// TIA Portal V17 export
// export: Created 2023-04-06T15:50:09.30215Z, ExportSetting WithDefaults, DisplayName Totally Integrated Automation Portal, DisplayVersion V17 Update 4, DisplayName TIA Portal Openness, DisplayVersion V17 Update 4, DisplayName TIA Portal Version Control Interface, DisplayVersion V17, DisplayName STEP 7 Professional, DisplayVersion V17 Update 4, DisplayName STEP 7 Safety, DisplayVersion V17, DisplayName WinCC Professional, DisplayVersion V17 Update 4
FUNCTION "LOGIC_PE_1" : Void   // FC7, LAD
{ S7_Optimized_Access := 'TRUE' }
VERSION : 0.1
// stored: AutoNumber true, IsIECCheckEnabled false, SetENOAutomatically false, UDAEnableTagReadback false
   VAR_TEMP
      rVac : Real;
   END_VAR
   VAR_TEMP   // added for the SCL form of the ladder/FBD networks
      _w1 : Bool;
      _w2 : Bool;
      _w3 : Bool;
   END_VAR
BEGIN

REGION Network 1: Write value of Password, P mode and Q mode - to check
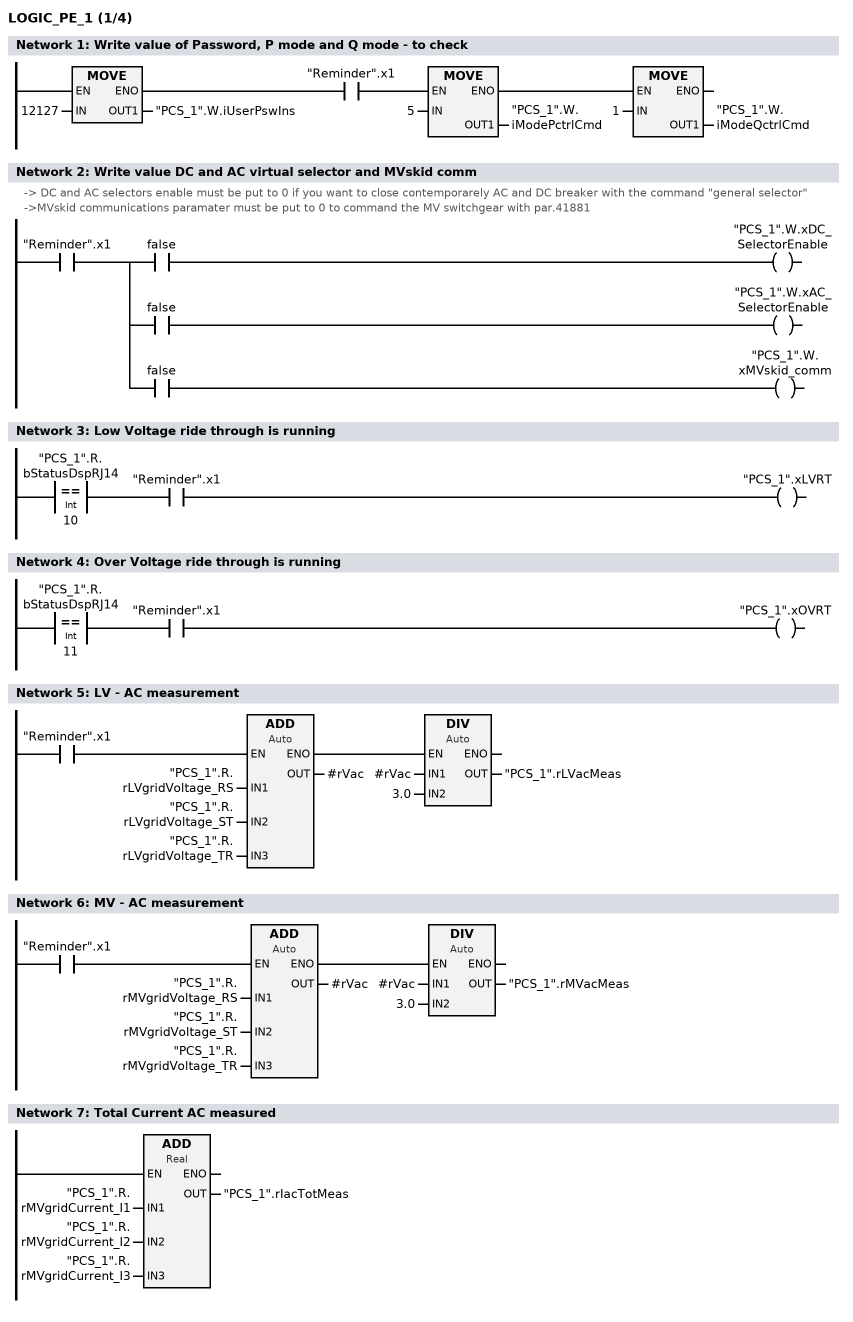
   RUNG wire#powerrail
      Move(in := 12127, out1 => "PCS_1".W.iUserPswIns)
      Contact( "Reminder".x1 )
      Move(in := 5, out1 => "PCS_1".W.iModePctrlCmd)
      Move(in := 1, out1 => "PCS_1".W.iModeQctrlCmd)
   END_RUNG
   // the same network as SCL:
   "PCS_1".W.iUserPswIns := 12127;
   IF "Reminder".x1 THEN
       "PCS_1".W.iModePctrlCmd := 5;
       "PCS_1".W.iModeQctrlCmd := 1;
   END_IF;
END_REGION

REGION Network 2: Write value DC and AC virtual selector and MVskid comm
   // -> DC and AC selectors enable must be put to 0 if you want to close contemporarely AC and DC breaker with the command "general selector"
   // ->MVskid communications paramater must be put to 0 to command the MV switchgear with par.41881
   RUNG wire#powerrail
      Contact( "Reminder".x1 )
      wire#w1
      Contact( false )
      Coil( "PCS_1".W.xDC_SelectorEnable )
   END_RUNG
   RUNG wire#w1
      Contact( false )
      Coil( "PCS_1".W.xAC_SelectorEnable )
   END_RUNG
   RUNG wire#w1
      Contact( false )
      Coil( "PCS_1".W.xMVskid_comm )
   END_RUNG
   // the same network as SCL:
   "PCS_1".W.xDC_SelectorEnable := "Reminder".x1 AND false;
   "PCS_1".W.xAC_SelectorEnable := "Reminder".x1 AND false;
   "PCS_1".W.xMVskid_comm := "Reminder".x1 AND false;
END_REGION

REGION Network 3: Low Voltage ride through is running
   RUNG wire#powerrail
      { S7_Templates := "SrcType := Int" } EQ_Contact(in1 := "PCS_1".R.bStatusDspRJ14, in2 := 10)
      Contact( "Reminder".x1 )
      Coil( "PCS_1".xLVRT )
   END_RUNG
   // the same network as SCL:
   "PCS_1".xLVRT := ("PCS_1".R.bStatusDspRJ14 = 10) AND "Reminder".x1;
END_REGION

REGION Network 4: Over Voltage ride through is running
   RUNG wire#powerrail
      { S7_Templates := "SrcType := Int" } EQ_Contact(in1 := "PCS_1".R.bStatusDspRJ14, in2 := 11)
      Contact( "Reminder".x1 )
      Coil( "PCS_1".xOVRT )
   END_RUNG
   // the same network as SCL:
   "PCS_1".xOVRT := ("PCS_1".R.bStatusDspRJ14 = 11) AND "Reminder".x1;
END_REGION

REGION Network 5: LV - AC measurement
   RUNG wire#powerrail
      Contact( "Reminder".x1 )
      Add(in1 := "PCS_1".R.rLVgridVoltage_RS, in2 := "PCS_1".R.rLVgridVoltage_ST, in3 := "PCS_1".R.rLVgridVoltage_TR, out => #rVac)
      Div(in1 := #rVac, in2 := 3.0, out => "PCS_1".rLVacMeas)
   END_RUNG
   // the same network as SCL:
   IF "Reminder".x1 THEN
       #rVac := "PCS_1".R.rLVgridVoltage_RS + "PCS_1".R.rLVgridVoltage_ST + "PCS_1".R.rLVgridVoltage_TR;
       "PCS_1".rLVacMeas := #rVac / 3.0;
   END_IF;
END_REGION

REGION Network 6: MV - AC measurement
   RUNG wire#powerrail
      Contact( "Reminder".x1 )
      Add(in1 := "PCS_1".R.rMVgridVoltage_RS, in2 := "PCS_1".R.rMVgridVoltage_ST, in3 := "PCS_1".R.rMVgridVoltage_TR, out => #rVac)
      Div(in1 := #rVac, in2 := 3.0, out => "PCS_1".rMVacMeas)
   END_RUNG
   // the same network as SCL:
   IF "Reminder".x1 THEN
       #rVac := "PCS_1".R.rMVgridVoltage_RS + "PCS_1".R.rMVgridVoltage_ST + "PCS_1".R.rMVgridVoltage_TR;
       "PCS_1".rMVacMeas := #rVac / 3.0;
   END_IF;
END_REGION

REGION Network 7: Total Current AC measured
   RUNG wire#powerrail
      { S7_Templates := "SrcType := Real" } Add(in1 := "PCS_1".R.rMVgridCurrent_I1, in2 := "PCS_1".R.rMVgridCurrent_I2, in3 := "PCS_1".R.rMVgridCurrent_I3, out => "PCS_1".rIacTotMeas)
   END_RUNG
   // the same network as SCL:
   "PCS_1".rIacTotMeas := "PCS_1".R.rMVgridCurrent_I1 + "PCS_1".R.rMVgridCurrent_I2 + "PCS_1".R.rMVgridCurrent_I3;
END_REGION

REGION Network 8: Inverter status
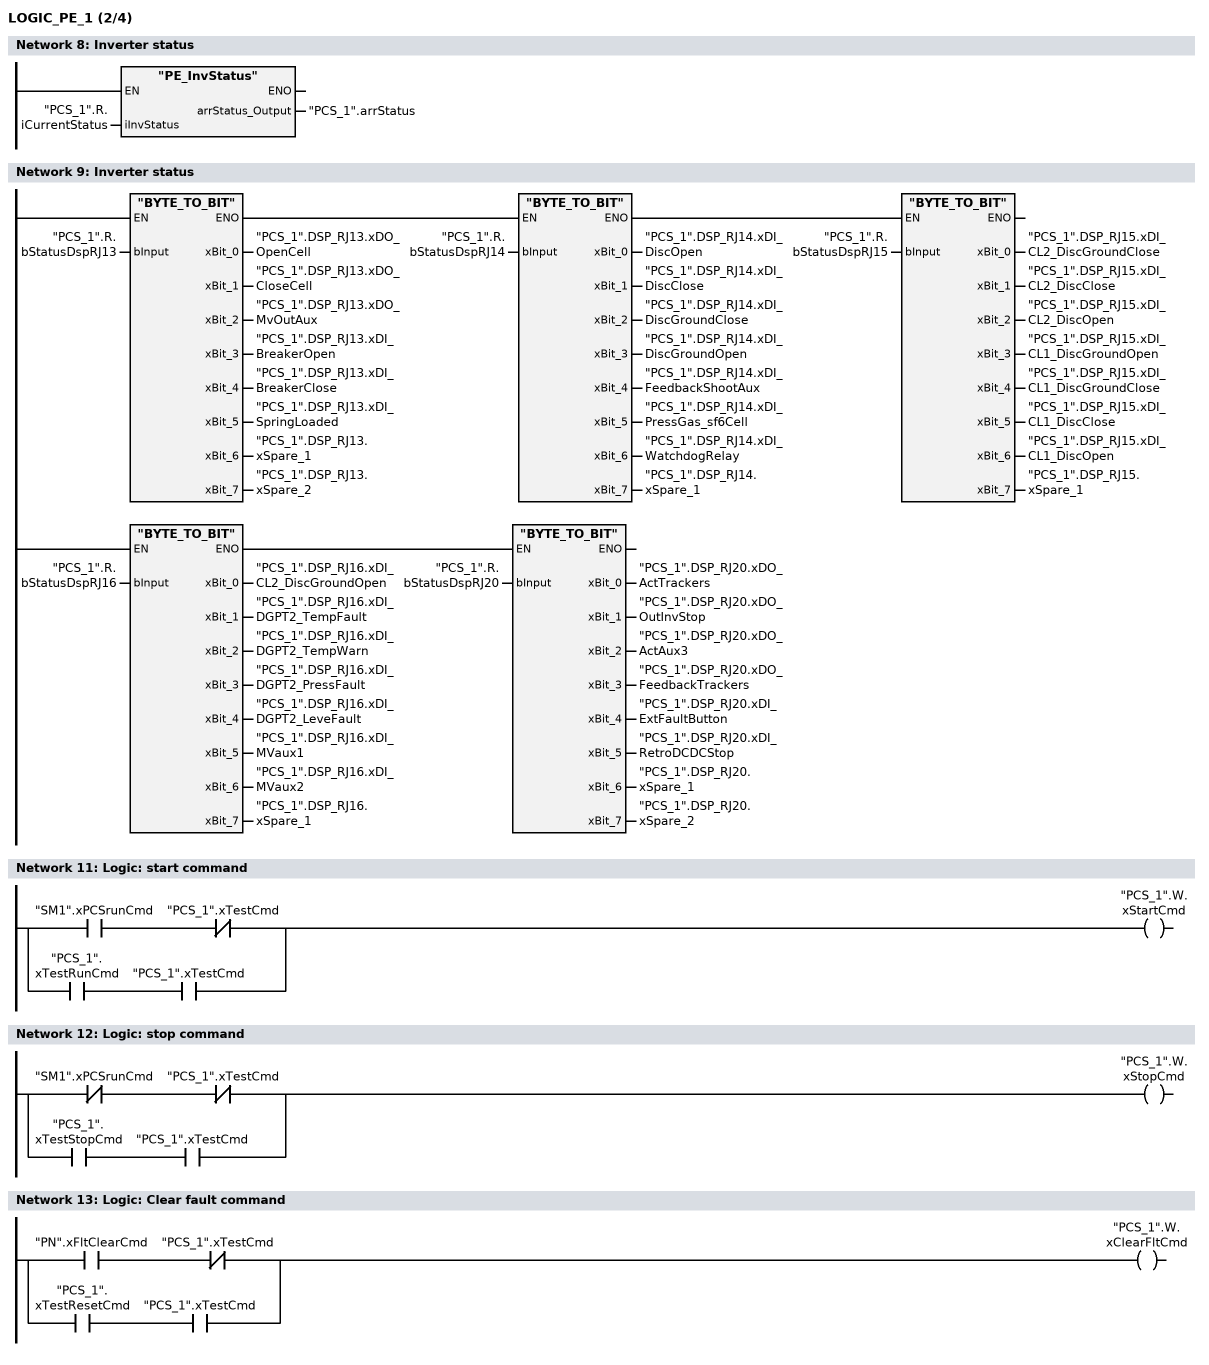
   RUNG wire#powerrail
      "PE_InvStatus"(iInvStatus := "PCS_1".R.iCurrentStatus, arrStatus_Output => "PCS_1".arrStatus)
   END_RUNG
   // the same network as SCL:
   "PE_InvStatus"(iInvStatus := "PCS_1".R.iCurrentStatus, arrStatus_Output => "PCS_1".arrStatus);
END_REGION

REGION Network 9: Inverter status
   RUNG wire#powerrail
      "BYTE_TO_BIT"(bInput := "PCS_1".R.bStatusDspRJ13, xBit_0 => "PCS_1".DSP_RJ13.xDO_OpenCell, xBit_1 => "PCS_1".DSP_RJ13.xDO_CloseCell, xBit_2 => "PCS_1".DSP_RJ13.xDO_MvOutAux, xBit_3 => "PCS_1".DSP_RJ13.xDI_BreakerOpen, xBit_4 => "PCS_1".DSP_RJ13.xDI_BreakerClose, xBit_5 => "PCS_1".DSP_RJ13.xDI_SpringLoaded, xBit_6 => "PCS_1".DSP_RJ13.xSpare_1, xBit_7 => "PCS_1".DSP_RJ13.xSpare_2)
      "BYTE_TO_BIT"(bInput := "PCS_1".R.bStatusDspRJ14, xBit_0 => "PCS_1".DSP_RJ14.xDI_DiscOpen, xBit_1 => "PCS_1".DSP_RJ14.xDI_DiscClose, xBit_2 => "PCS_1".DSP_RJ14.xDI_DiscGroundClose, xBit_3 => "PCS_1".DSP_RJ14.xDI_DiscGroundOpen, xBit_4 => "PCS_1".DSP_RJ14.xDI_FeedbackShootAux, xBit_5 => "PCS_1".DSP_RJ14.xDI_PressGas_sf6Cell, xBit_6 => "PCS_1".DSP_RJ14.xDI_WatchdogRelay, xBit_7 => "PCS_1".DSP_RJ14.xSpare_1)
      "BYTE_TO_BIT"(bInput := "PCS_1".R.bStatusDspRJ15, xBit_0 => "PCS_1".DSP_RJ15.xDI_CL2_DiscGroundClose, xBit_1 => "PCS_1".DSP_RJ15.xDI_CL2_DiscClose, xBit_2 => "PCS_1".DSP_RJ15.xDI_CL2_DiscOpen, xBit_3 => "PCS_1".DSP_RJ15.xDI_CL1_DiscGroundOpen, xBit_4 => "PCS_1".DSP_RJ15.xDI_CL1_DiscGroundClose, xBit_5 => "PCS_1".DSP_RJ15.xDI_CL1_DiscClose, xBit_6 => "PCS_1".DSP_RJ15.xDI_CL1_DiscOpen, xBit_7 => "PCS_1".DSP_RJ15.xSpare_1)
   END_RUNG
   RUNG wire#powerrail
      "BYTE_TO_BIT"(bInput := "PCS_1".R.bStatusDspRJ16, xBit_0 => "PCS_1".DSP_RJ16.xDI_CL2_DiscGroundOpen, xBit_1 => "PCS_1".DSP_RJ16.xDI_DGPT2_TempFault, xBit_2 => "PCS_1".DSP_RJ16.xDI_DGPT2_TempWarn, xBit_3 => "PCS_1".DSP_RJ16.xDI_DGPT2_PressFault, xBit_4 => "PCS_1".DSP_RJ16.xDI_DGPT2_LeveFault, xBit_5 => "PCS_1".DSP_RJ16.xDI_MVaux1, xBit_6 => "PCS_1".DSP_RJ16.xDI_MVaux2, xBit_7 => "PCS_1".DSP_RJ16.xSpare_1)
      "BYTE_TO_BIT"(bInput := "PCS_1".R.bStatusDspRJ20, xBit_0 => "PCS_1".DSP_RJ20.xDO_ActTrackers, xBit_1 => "PCS_1".DSP_RJ20.xDO_OutInvStop, xBit_2 => "PCS_1".DSP_RJ20.xDO_ActAux3, xBit_3 => "PCS_1".DSP_RJ20.xDO_FeedbackTrackers, xBit_4 => "PCS_1".DSP_RJ20.xDI_ExtFaultButton, xBit_5 => "PCS_1".DSP_RJ20.xDI_RetroDCDCStop, xBit_6 => "PCS_1".DSP_RJ20.xSpare_1, xBit_7 => "PCS_1".DSP_RJ20.xSpare_2)
   END_RUNG
   // the same network as SCL:
   "BYTE_TO_BIT"(bInput := "PCS_1".R.bStatusDspRJ13,
                 xBit_0 => "PCS_1".DSP_RJ13.xDO_OpenCell,
                 xBit_1 => "PCS_1".DSP_RJ13.xDO_CloseCell,
                 xBit_2 => "PCS_1".DSP_RJ13.xDO_MvOutAux,
                 xBit_3 => "PCS_1".DSP_RJ13.xDI_BreakerOpen,
                 xBit_4 => "PCS_1".DSP_RJ13.xDI_BreakerClose,
                 xBit_5 => "PCS_1".DSP_RJ13.xDI_SpringLoaded,
                 xBit_6 => "PCS_1".DSP_RJ13.xSpare_1,
                 xBit_7 => "PCS_1".DSP_RJ13.xSpare_2,
                 ENO => #_w1);
   "BYTE_TO_BIT"(EN := #_w1,
                 bInput := "PCS_1".R.bStatusDspRJ14,
                 xBit_0 => "PCS_1".DSP_RJ14.xDI_DiscOpen,
                 xBit_1 => "PCS_1".DSP_RJ14.xDI_DiscClose,
                 xBit_2 => "PCS_1".DSP_RJ14.xDI_DiscGroundClose,
                 xBit_3 => "PCS_1".DSP_RJ14.xDI_DiscGroundOpen,
                 xBit_4 => "PCS_1".DSP_RJ14.xDI_FeedbackShootAux,
                 xBit_5 => "PCS_1".DSP_RJ14.xDI_PressGas_sf6Cell,
                 xBit_6 => "PCS_1".DSP_RJ14.xDI_WatchdogRelay,
                 xBit_7 => "PCS_1".DSP_RJ14.xSpare_1,
                 ENO => #_w2);
   IF #_w2 THEN
       "BYTE_TO_BIT"(bInput := "PCS_1".R.bStatusDspRJ15,
                     xBit_0 => "PCS_1".DSP_RJ15.xDI_CL2_DiscGroundClose,
                     xBit_1 => "PCS_1".DSP_RJ15.xDI_CL2_DiscClose,
                     xBit_2 => "PCS_1".DSP_RJ15.xDI_CL2_DiscOpen,
                     xBit_3 => "PCS_1".DSP_RJ15.xDI_CL1_DiscGroundOpen,
                     xBit_4 => "PCS_1".DSP_RJ15.xDI_CL1_DiscGroundClose,
                     xBit_5 => "PCS_1".DSP_RJ15.xDI_CL1_DiscClose,
                     xBit_6 => "PCS_1".DSP_RJ15.xDI_CL1_DiscOpen,
                     xBit_7 => "PCS_1".DSP_RJ15.xSpare_1);
   END_IF;
   "BYTE_TO_BIT"(bInput := "PCS_1".R.bStatusDspRJ16,
                 xBit_0 => "PCS_1".DSP_RJ16.xDI_CL2_DiscGroundOpen,
                 xBit_1 => "PCS_1".DSP_RJ16.xDI_DGPT2_TempFault,
                 xBit_2 => "PCS_1".DSP_RJ16.xDI_DGPT2_TempWarn,
                 xBit_3 => "PCS_1".DSP_RJ16.xDI_DGPT2_PressFault,
                 xBit_4 => "PCS_1".DSP_RJ16.xDI_DGPT2_LeveFault,
                 xBit_5 => "PCS_1".DSP_RJ16.xDI_MVaux1,
                 xBit_6 => "PCS_1".DSP_RJ16.xDI_MVaux2,
                 xBit_7 => "PCS_1".DSP_RJ16.xSpare_1,
                 ENO => #_w3);
   IF #_w3 THEN
       "BYTE_TO_BIT"(bInput := "PCS_1".R.bStatusDspRJ20,
                     xBit_0 => "PCS_1".DSP_RJ20.xDO_ActTrackers,
                     xBit_1 => "PCS_1".DSP_RJ20.xDO_OutInvStop,
                     xBit_2 => "PCS_1".DSP_RJ20.xDO_ActAux3,
                     xBit_3 => "PCS_1".DSP_RJ20.xDO_FeedbackTrackers,
                     xBit_4 => "PCS_1".DSP_RJ20.xDI_ExtFaultButton,
                     xBit_5 => "PCS_1".DSP_RJ20.xDI_RetroDCDCStop,
                     xBit_6 => "PCS_1".DSP_RJ20.xSpare_1,
                     xBit_7 => "PCS_1".DSP_RJ20.xSpare_2);
   END_IF;
END_REGION

REGION Network 11: Logic: start command
   RUNG wire#powerrail
      Contact( "SM1".xPCSrunCmd )
      I_Contact( "PCS_1".xTestCmd )
      wire#w1
      Coil( "PCS_1".W.xStartCmd )
   END_RUNG
   RUNG wire#powerrail
      Contact( "PCS_1".xTestRunCmd )
      Contact( "PCS_1".xTestCmd )
   END_RUNG wire#w1
   // the same network as SCL:
   "PCS_1".W.xStartCmd := ("SM1".xPCSrunCmd AND NOT "PCS_1".xTestCmd) OR ("PCS_1".xTestRunCmd AND "PCS_1".xTestCmd);
END_REGION

REGION Network 12: Logic: stop command
   RUNG wire#powerrail
      I_Contact( "SM1".xPCSrunCmd )
      I_Contact( "PCS_1".xTestCmd )
      wire#w1
      Coil( "PCS_1".W.xStopCmd )
   END_RUNG
   RUNG wire#powerrail
      Contact( "PCS_1".xTestStopCmd )
      Contact( "PCS_1".xTestCmd )
   END_RUNG wire#w1
   // the same network as SCL:
   "PCS_1".W.xStopCmd := (NOT "SM1".xPCSrunCmd AND NOT "PCS_1".xTestCmd) OR ("PCS_1".xTestStopCmd AND "PCS_1".xTestCmd);
END_REGION

REGION Network 13: Logic: Clear fault command
   RUNG wire#powerrail
      Contact( "PN".xFltClearCmd )
      I_Contact( "PCS_1".xTestCmd )
      wire#w1
      Coil( "PCS_1".W.xClearFltCmd )
   END_RUNG
   RUNG wire#powerrail
      Contact( "PCS_1".xTestResetCmd )
      Contact( "PCS_1".xTestCmd )
   END_RUNG wire#w1
   // the same network as SCL:
   "PCS_1".W.xClearFltCmd := ("PN".xFltClearCmd AND NOT "PCS_1".xTestCmd) OR ("PCS_1".xTestResetCmd AND "PCS_1".xTestCmd);
END_REGION

REGION Network 14: Logic : PPC enable command
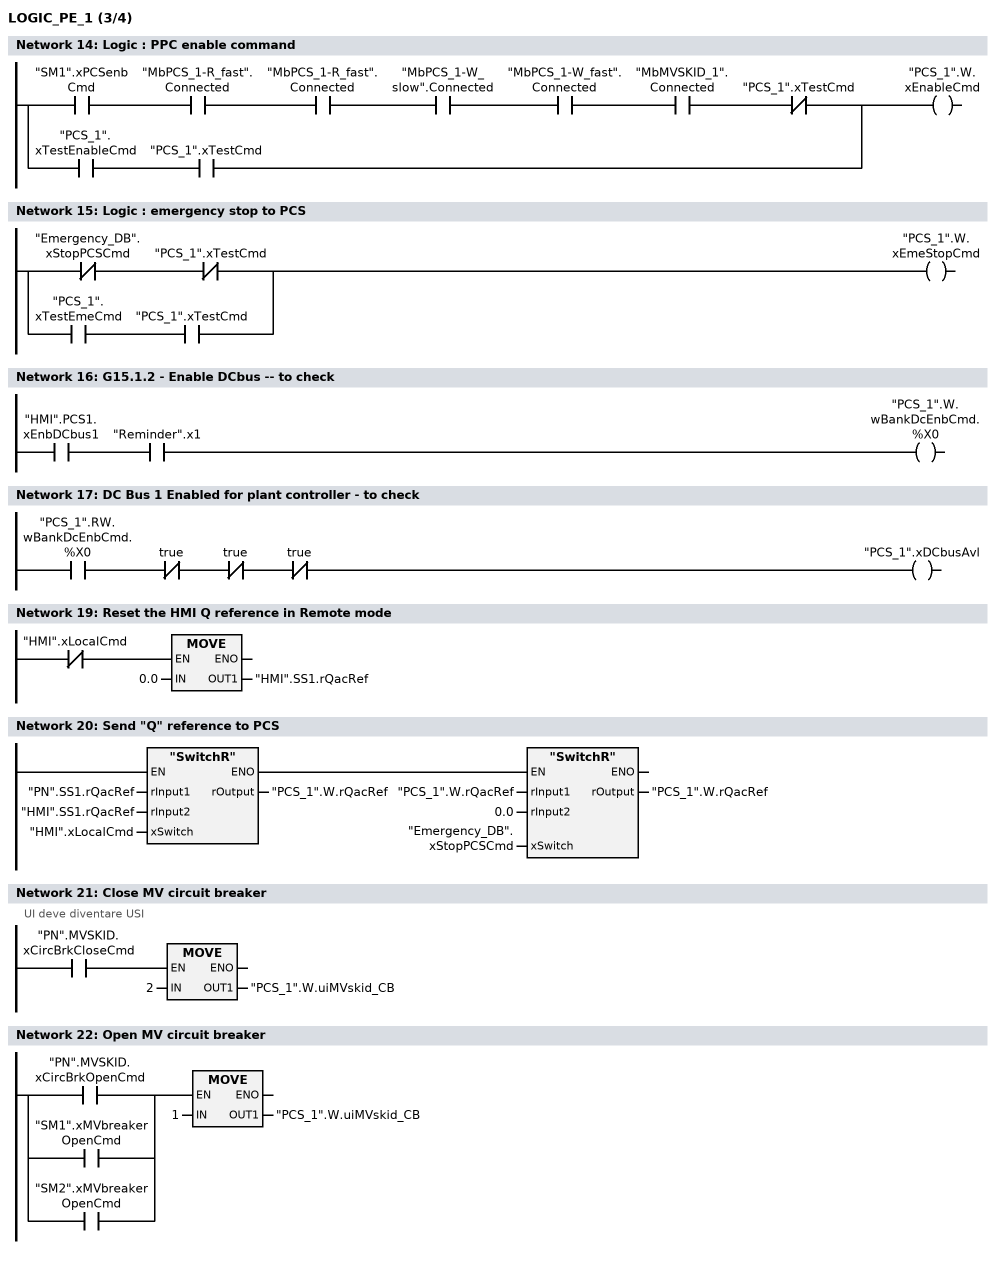
   RUNG wire#powerrail
      Contact( "SM1".xPCSenbCmd )
      Contact( "MbPCS_1-R_fast".Connected )
      Contact( "MbPCS_1-R_fast".Connected )
      Contact( "MbPCS_1-W_slow".Connected )
      Contact( "MbPCS_1-W_fast".Connected )
      Contact( "MbMVSKID_1".Connected )
      I_Contact( "PCS_1".xTestCmd )
      wire#w1
      Coil( "PCS_1".W.xEnableCmd )
   END_RUNG
   RUNG wire#powerrail
      Contact( "PCS_1".xTestEnableCmd )
      Contact( "PCS_1".xTestCmd )
   END_RUNG wire#w1
   // the same network as SCL:
   "PCS_1".W.xEnableCmd := ("SM1".xPCSenbCmd AND "MbPCS_1-R_fast".Connected AND "MbPCS_1-R_fast".Connected AND "MbPCS_1-W_slow".Connected AND "MbPCS_1-W_fast".Connected AND "MbMVSKID_1".Connected AND NOT "PCS_1".xTestCmd) OR ("PCS_1".xTestEnableCmd AND "PCS_1".xTestCmd);
END_REGION

REGION Network 15: Logic : emergency stop to PCS
   RUNG wire#powerrail
      I_Contact( "Emergency_DB".xStopPCSCmd )
      I_Contact( "PCS_1".xTestCmd )
      wire#w1
      Coil( "PCS_1".W.xEmeStopCmd )
   END_RUNG
   RUNG wire#powerrail
      Contact( "PCS_1".xTestEmeCmd )
      Contact( "PCS_1".xTestCmd )
   END_RUNG wire#w1
   // the same network as SCL:
   "PCS_1".W.xEmeStopCmd := (NOT "Emergency_DB".xStopPCSCmd AND NOT "PCS_1".xTestCmd) OR ("PCS_1".xTestEmeCmd AND "PCS_1".xTestCmd);
END_REGION

REGION Network 16: G15.1.2 - Enable DCbus -- to check
   RUNG wire#powerrail
      Contact( "HMI".PCS1.xEnbDCbus1 )
      Contact( "Reminder".x1 )
      Coil( "PCS_1".W.wBankDcEnbCmd.%X0 )
   END_RUNG
   // the same network as SCL:
   "PCS_1".W.wBankDcEnbCmd.%X0 := "HMI".PCS1.xEnbDCbus1 AND "Reminder".x1;
END_REGION

REGION Network 17: DC Bus 1 Enabled for plant controller - to check
   RUNG wire#powerrail
      Contact( "PCS_1".RW.wBankDcEnbCmd.%X0 )
      I_Contact( true )
      I_Contact( true )
      I_Contact( true )
      Coil( "PCS_1".xDCbusAvl )
   END_RUNG
   // the same network as SCL:
   "PCS_1".xDCbusAvl := "PCS_1".RW.wBankDcEnbCmd.%X0 AND NOT true AND NOT true AND NOT true;
END_REGION

REGION Network 19: Reset the HMI Q reference in Remote mode
   RUNG wire#powerrail
      I_Contact( "HMI".xLocalCmd )
      Move(in := 0.0, out1 => "HMI".SS1.rQacRef)
   END_RUNG
   // the same network as SCL:
   IF NOT "HMI".xLocalCmd THEN "HMI".SS1.rQacRef := 0.0; END_IF;
END_REGION

REGION Network 20: Send "Q" reference to PCS
   RUNG wire#powerrail
      "SwitchR"(rInput1 := "PN".SS1.rQacRef, rInput2 := "HMI".SS1.rQacRef, xSwitch := "HMI".xLocalCmd, rOutput => "PCS_1".W.rQacRef)
      "SwitchR"(rInput1 := "PCS_1".W.rQacRef, rInput2 := 0.0, xSwitch := "Emergency_DB".xStopPCSCmd, rOutput => "PCS_1".W.rQacRef)
   END_RUNG
   // the same network as SCL:
   "SwitchR"(rInput1 := "PN".SS1.rQacRef,
             rInput2 := "HMI".SS1.rQacRef,
             xSwitch := "HMI".xLocalCmd,
             rOutput => "PCS_1".W.rQacRef,
             ENO => #_w1);
   IF #_w1 THEN
       "SwitchR"(rInput1 := "PCS_1".W.rQacRef,
                 rInput2 := 0.0,
                 xSwitch := "Emergency_DB".xStopPCSCmd,
                 rOutput => "PCS_1".W.rQacRef);
   END_IF;
END_REGION

REGION Network 21: Close MV circuit breaker
   // UI deve diventare USI
   RUNG wire#powerrail
      Contact( "PN".MVSKID.xCircBrkCloseCmd )
      Move(in := 2, out1 => "PCS_1".W.uiMVskid_CB)
   END_RUNG
   // the same network as SCL:
   IF "PN".MVSKID.xCircBrkCloseCmd THEN "PCS_1".W.uiMVskid_CB := 2; END_IF;
END_REGION

REGION Network 22: Open MV circuit breaker
   RUNG wire#powerrail
      Contact( "PN".MVSKID.xCircBrkOpenCmd )
      wire#w1
      Move(in := 1, out1 => "PCS_1".W.uiMVskid_CB)
   END_RUNG
   RUNG wire#powerrail
      Contact( "SM1".xMVbreakerOpenCmd )
   END_RUNG wire#w1
   RUNG wire#powerrail
      Contact( "SM2".xMVbreakerOpenCmd )
   END_RUNG wire#w1
   // the same network as SCL:
   IF "PN".MVSKID.xCircBrkOpenCmd OR "SM1".xMVbreakerOpenCmd OR "SM2".xMVbreakerOpenCmd THEN
       "PCS_1".W.uiMVskid_CB := 1;
   END_IF;
END_REGION

REGION Network 23: MV SKID Fault
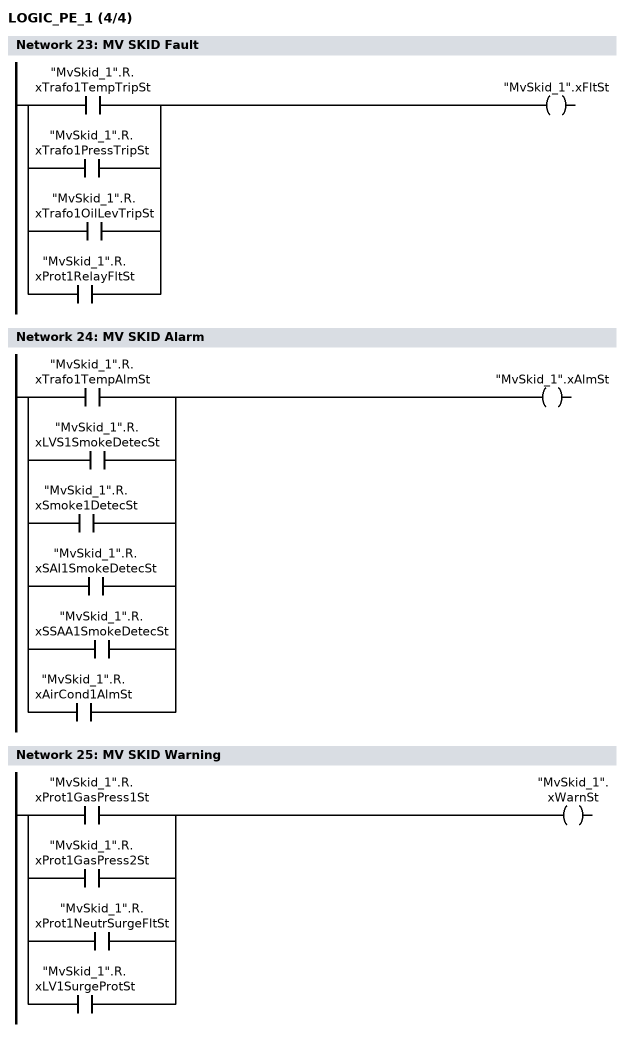
   RUNG wire#powerrail
      Contact( "MvSkid_1".R.xTrafo1TempTripSt )
      wire#w1
      Coil( "MvSkid_1".xFltSt )
   END_RUNG
   RUNG wire#powerrail
      Contact( "MvSkid_1".R.xTrafo1PressTripSt )
   END_RUNG wire#w1
   RUNG wire#powerrail
      Contact( "MvSkid_1".R.xTrafo1OilLevTripSt )
   END_RUNG wire#w1
   RUNG wire#powerrail
      Contact( "MvSkid_1".R.xProt1RelayFltSt )
   END_RUNG wire#w1
   // the same network as SCL:
   "MvSkid_1".xFltSt := "MvSkid_1".R.xTrafo1TempTripSt OR "MvSkid_1".R.xTrafo1PressTripSt OR "MvSkid_1".R.xTrafo1OilLevTripSt OR "MvSkid_1".R.xProt1RelayFltSt;
END_REGION

REGION Network 24: MV SKID Alarm
   RUNG wire#powerrail
      Contact( "MvSkid_1".R.xTrafo1TempAlmSt )
      wire#w1
      Coil( "MvSkid_1".xAlmSt )
   END_RUNG
   RUNG wire#powerrail
      Contact( "MvSkid_1".R.xLVS1SmokeDetecSt )
   END_RUNG wire#w1
   RUNG wire#powerrail
      Contact( "MvSkid_1".R.xSmoke1DetecSt )
   END_RUNG wire#w1
   RUNG wire#powerrail
      Contact( "MvSkid_1".R.xSAI1SmokeDetecSt )
   END_RUNG wire#w1
   RUNG wire#powerrail
      Contact( "MvSkid_1".R.xSSAA1SmokeDetecSt )
   END_RUNG wire#w1
   RUNG wire#powerrail
      Contact( "MvSkid_1".R.xAirCond1AlmSt )
   END_RUNG wire#w1
   // the same network as SCL:
   "MvSkid_1".xAlmSt := "MvSkid_1".R.xTrafo1TempAlmSt OR "MvSkid_1".R.xLVS1SmokeDetecSt OR "MvSkid_1".R.xSmoke1DetecSt OR "MvSkid_1".R.xSAI1SmokeDetecSt OR "MvSkid_1".R.xSSAA1SmokeDetecSt OR "MvSkid_1".R.xAirCond1AlmSt;
END_REGION

REGION Network 25: MV SKID Warning
   RUNG wire#powerrail
      Contact( "MvSkid_1".R.xProt1GasPress1St )
      wire#w1
      Coil( "MvSkid_1".xWarnSt )
   END_RUNG
   RUNG wire#powerrail
      Contact( "MvSkid_1".R.xProt1GasPress2St )
   END_RUNG wire#w1
   RUNG wire#powerrail
      Contact( "MvSkid_1".R.xProt1NeutrSurgeFltSt )
   END_RUNG wire#w1
   RUNG wire#powerrail
      Contact( "MvSkid_1".R.xLV1SurgeProtSt )
   END_RUNG wire#w1
   // the same network as SCL:
   "MvSkid_1".xWarnSt := "MvSkid_1".R.xProt1GasPress1St OR "MvSkid_1".R.xProt1GasPress2St OR "MvSkid_1".R.xProt1NeutrSurgeFltSt OR "MvSkid_1".R.xLV1SurgeProtSt;
END_REGION

REGION Network 26 (SCL): MV SKID Line Disconnector & Breaker Status
   "MvSkid_1".wLine1DiscSt.%X0 := "MvSkid_1".R.xLine1DiscOpenSt;
   "MvSkid_1".wLine1DiscSt.%X1 := "MvSkid_1".R.xLine1DiscCloseSt;
   "MvSkid_1".wLine1DiscSt.%X2 := "MvSkid_1".R.xLine1GndCloseSt;

   "MvSkid_1".wLine2DiscSt.%X0 := "MvSkid_1".R.xLine2DiscOpenSt;
   "MvSkid_1".wLine2DiscSt.%X1 := "MvSkid_1".R.xLine2DiscCloseSt;
   "MvSkid_1".wLine2DiscSt.%X2 := "MvSkid_1".R.xLine2GndCloseSt;

   "MvSkid_1".wProt1DiscSt.%X0 := "MvSkid_1".R.xProt1DiscOpenSt;
   "MvSkid_1".wProt1DiscSt.%X1 := "MvSkid_1".R.xProt1DiscCloseSt;
   "MvSkid_1".wProt1DiscSt.%X2 := "MvSkid_1".R.xProt1GndCloseSt;

   "MvSkid_1".wProt1CircBrkSt.%X0 := "MvSkid_1".R.xProt1CircBrkOpenSt;
   "MvSkid_1".wProt1CircBrkSt.%X1 := "MvSkid_1".R.xProt1CircBrkCloseSt;
END_REGION
END_FUNCTION
